// TIA Portal V17 export
// export: Created 2022-06-27T13:57:17.7614963Z, ExportSetting WithDefaults, DisplayName Totally Integrated Automation Portal, DisplayVersion V17 Update 3, DisplayName TIA Portal Openness, DisplayVersion V17 Update 3, DisplayName TIA Portal Version Control Interface, DisplayVersion V17, DisplayName SINAMICS Startdrive Advanced, DisplayVersion V17 Update1, DisplayName SINAMICS Startdrive G110M, G120, G120C, G120D, G120P, G115D, DisplayVersion V17 Update1, DisplayName SINAMICS Startdrive G130, G150, S120, S150, SINAMICS MV, S210, DisplayVersion V17 Update1, DisplayName STEP 7 Professional, DisplayVersion V17 Update 3, DisplayName STEP 7 Safety, DisplayVersion V17, DisplayName WinCC UA Professional, DisplayVersion V17 Update 3
FUNCTION_BLOCK "S032_DUMPER_VALVES"   // FB32, LAD
{ S7_Optimized_Access := 'TRUE' }
VERSION : 0.1
// stored: AutoNumber false, IsIECCheckEnabled false, IsRetainMemResEnabled false, MemoryReserve 100, SetENOAutomatically false, UDAEnableTagReadback false
BEGIN

REGION Network 1: FY86-2E - Hot Air Dumper Chamber 1 - Automatic on and off
END_REGION

REGION Network 2: FY86-2E - Hot Air Dumper Chamber 1 - Interlocks
END_REGION

REGION Network 3: FY86-2E - Hot Air Dumper Chamber 1 - Setpoint
END_REGION

REGION Network 4: FY86-2E - Hot Air Dumper Chamber 1 - Force Conditions
END_REGION

REGION Network 5: FY86-2E - Hot Air Dumper Chamber 1 - Temperature Control (PID)
END_REGION

REGION Network 6: FY86-2E - Hot Air Dumper Chamber 1 - Valve Function Call
END_REGION

REGION Network 8: FY86-4E - Ambient Air Dumper Chamber 1 - Automatic on and off
END_REGION

REGION Network 9: FY86-4E - Ambient Air Dumper Chamber 1 - Interlocks
END_REGION

REGION Network 10: FY86-4E - Ambient Air Dumper Chamber 1 - Setpoint
END_REGION

REGION Network 11: FY86-4E - Ambient Air Dumper Chamber 1 - Force Conditions
END_REGION

REGION Network 12: FY86-4E - Ambient Air Dumper Chamber 1 - Temperature Control (PID)
END_REGION

REGION Network 13: FY86-4E - Ambient Air Dumper Chamber 1 - Valve Function Call
END_REGION

REGION Network 15: FY87-2E - Hot Air Dumper Chamber 2 - Automatic on and off
END_REGION

REGION Network 16: FY87-2E - Hot Air Dumper Chamber 2 - Interlocks
END_REGION

REGION Network 17: FY87-2E - Hot Air Dumper Chamber 2 - Setpoint
END_REGION

REGION Network 18: FY87-2E - Hot Air Dumper Chamber 2 - Force Conditions
END_REGION

REGION Network 19: FY87-2E - Hot Air Dumper Chamber 2 - Temperature Control (PID)
END_REGION

REGION Network 20: FY87-2E - Hot Air Dumper Chamber 2 - Valve Function Call
END_REGION

REGION Network 22: FY87-4E - Ambient Air Dumper Chamber 2 - Automatic on and off
END_REGION

REGION Network 23: FY87-4E - Ambient Air Dumper Chamber 2 - Interlocks
END_REGION

REGION Network 24: FY87-4E - Ambient Air Dumper Chamber 2 - Setpoint
END_REGION

REGION Network 25: FY87-4E - Ambient Air Dumper Chamber 2 - Force Conditions
END_REGION

REGION Network 26: FY87-4E - Ambient Air Dumper Chamber 2 - Temperature Control (PID)
END_REGION

REGION Network 27: FY87-4E - Ambient Air Dumper Chamber 2 - Valve Function Call
END_REGION
END_FUNCTION_BLOCK
